KUKA KRL program: PickPlace01.src, PickPlace01.dat

--- PickPlace01.src ---
&ACCESS RVP
&REL 1
&COMMENT Pick and place demo
DEF PickPlace01()
  ;FOLD INI
    ;FOLD BASISTECH INI
      BAS(#INITMOV, 0)
    ;ENDFOLD
  ;ENDFOLD

  PTP HOME Vel=100% DEFAULT

  ;FOLD PTP P1 Vel=100% PDAT1 Tool[1] Base[0]
    PTP P1 Vel=100% PDAT1 Tool[1] Base[0]
  ;ENDFOLD

  ;FOLD LIN P2 Vel=2m/s CPDAT1 Tool[1] Base[0]
    LIN P2 Vel=2m/s CPDAT1 Tool[1] Base[0]
  ;ENDFOLD

  ;FOLD GRIPPER CLOSE
    $OUT[1] = TRUE
    WAIT SEC 0.5
  ;ENDFOLD

  ;FOLD PTP P3 Vel=100% PDAT2 Tool[1] Base[0]
    PTP P3 Vel=100% PDAT2 Tool[1] Base[0]
  ;ENDFOLD

  ;FOLD GRIPPER OPEN
    $OUT[1] = FALSE
    WAIT SEC 0.5
  ;ENDFOLD

  PTP HOME Vel=100% DEFAULT

END

--- PickPlace01.dat ---
DEFDAT PickPlace01
  ;FOLD EXTERNAL DECLARATIONS; %{PE}
  ;ENDFOLD

  DECL E6POS HOME={A1 0.0, A2 -90.0, A3 90.0, A4 0.0, A5 0.0, A6 0.0}
  DECL E6POS P1={X 500.0, Y 200.0, Z 400.0, A 0.0, B 90.0, C 0.0, S 2, T 10}
  DECL E6POS P2={X 500.0, Y 200.0, Z 200.0, A 0.0, B 90.0, C 0.0, S 2, T 10}
  DECL E6POS P3={X 500.0, Y -200.0, Z 400.0, A 0.0, B 90.0, C 0.0, S 2, T 10}

ENDDAT
